INTERFACE I_Outputs
VAR
	n_temp_speed:REAL;
	n_target_speed:REAL;
	
	
	
END_VAR

END_INTERFACE

(* stored: Version 1.1.0.1, ProductVersion 3.1.4024.11
   Itf I_Outputs: Id {ffac5a95-3400-4dee-9e8d-0287965b5ddb} *)
